(* PLC project PLC, Beckhoff Automation GmbH TwinCAT PLC Control 3.5.13.21 *)
(* stored: creationDateTime 2022-06-22T22:53:39.582356, modificationDateTime 2022-06-22T22:53:39.582356 *)

FUNCTION_BLOCK BCD_TO_DWORD
VAR_INPUT
	en: BOOL;
	bin: DWORD;
END_VAR
VAR_OUTPUT
	eno: BOOL;
	err: BOOL;
	wout: DWORD;
END_VAR
VAR
	digit: INT;
	n: DWORD;
END_VAR

            err := FALSE;
wout := 0;

IF en THEN
	FOR digit := 0 TO 7 DO
		n := SHR(bin AND SHL(16#F, digit * 4), digit * 4);
		IF n > 9 THEN
			err := TRUE;
			RETURN;
		END_IF
		wout := wout + n * LREAL_TO_DWORD(EXPT(10, digit));
	END_FOR
	eno := TRUE;
ELSE
	eno := FALSE;
END_IF
          
END_FUNCTION_BLOCK
